FUNCTION_BLOCK MoveMod IMPLEMENTS I_MoveMod
VAR
	mcMoveMod : MC_MoveModulo;
END_VAR
VAR_IN_OUT
	Axis : AXIS_REF;
END_VAR

mcMoveMod(Axis := Axis);

PROPERTY Acceleration : MC_LREAL
GET
Acceleration := mcMoveMod.Acceleration;
END_GET
SET
mcMoveMod.Acceleration := Acceleration;
END_SET
END_PROPERTY

PROPERTY BufferMode : MC_Buffermode
GET
BufferMode := mcMoveMod.BufferMode;
END_GET
SET
mcMoveMod.BufferMode := BufferMode;
END_SET
END_PROPERTY

PROPERTY Busy : BOOL
GET
Busy := mcMoveMod.Busy;
END_GET
END_PROPERTY

PROPERTY Deceleration : MC_LREAL
GET
Deceleration := mcMoveMod.Deceleration;
END_GET
SET
mcMoveMod.Deceleration := Deceleration;
END_SET
END_PROPERTY

PROPERTY Done : BOOL
GET
Done := mcMoveMod.Done;
END_GET
END_PROPERTY

PROPERTY Error : BOOL
GET
Error := mcMoveMod.Error;
END_GET
END_PROPERTY

PROPERTY Execute : BOOL
GET
Execute := mcMoveMod.Execute;
END_GET
SET
mcMoveMod.Execute := Execute;
END_SET
END_PROPERTY

PROPERTY Jerk : MC_LREAL
GET
Jerk := mcMoveMod.Jerk;
END_GET
SET
mcMoveMod.Jerk := Jerk;
END_SET
END_PROPERTY

PROPERTY Position : MC_LREAL
GET
Position := mcMoveMod.Position;
END_GET
SET
mcMoveMod.Position := Position;
END_SET
END_PROPERTY

PROPERTY Velocity : MC_LREAL
GET
Velocity := mcMoveMod.Velocity;
END_GET
SET
mcMoveMod.Velocity := Velocity;
END_SET
END_PROPERTY

END_FUNCTION_BLOCK

(* stored: Version 1.1.0.1
   POU MoveMod: Id {1bfd3278-afcc-4c3c-bae2-f1c6b30d8866}, SpecialFunc None
   Property Acceleration: Id {0d596a7e-59a4-4ff1-b65d-5147cb01f504}
   Get Get: Id {fa6a6f62-d27e-4c07-bef8-33f473fbbcdf}
   Set Set: Id {bec1acfe-50dd-4e03-b13f-0075cdea64fe}
   Property BufferMode: Id {383aa336-aecf-4729-be5a-4928a876364b}
   Get Get: Id {476d401d-a9d7-49ed-8580-9ec8f334d596}
   Set Set: Id {c3669d7b-b91c-4b87-9cbc-09ce1123b73b}
   Property Busy: Id {4f906338-2c35-4182-8130-4b088126df2e}
   Get Get: Id {e2677317-bb42-4496-8737-fc1a199be176}
   Property Deceleration: Id {23702022-baef-491d-8e8a-39565a6c0db1}
   Get Get: Id {41cffb6c-884b-4af2-97ef-8c9ceeb6ee4d}
   Set Set: Id {aeb20737-4404-4eed-9314-f137f39cb149}
   Property Done: Id {9d49c45d-888f-4f5f-abe7-ea7dcff52795}
   Get Get: Id {4d1d556f-75ae-457f-a49c-79d62f4cc6e4}
   Property Error: Id {a092da43-f5c5-4fc3-9ad4-9f21a689b071}
   Get Get: Id {ec2bddf4-5474-4cf0-86db-2bcd939479ee}
   Property Execute: Id {6729b1eb-82a3-4bec-ac1a-aed1fbe49052}
   Get Get: Id {7614de87-20d3-4733-995e-df3b16396c9e}
   Set Set: Id {c7fb56e5-7530-4953-974a-30bb8a162548}
   Property Jerk: Id {1dfb9313-e978-46a2-a93b-14d64bbdd93e}
   Get Get: Id {dd16343b-3036-4d2c-a8eb-64bab3590434}
   Set Set: Id {ee01a914-c076-4eb4-97d0-bce7cca76172}
   Property Position: Id {7c12b022-2f2b-4f2b-b8ee-e4ff0a495548}
   Get Get: Id {39ffb0f6-b656-445c-a80a-557075a93232}
   Set Set: Id {9adab8d2-9008-44dc-9e2c-3d171b4e9df4}
   Property Velocity: Id {121742a5-e664-4c8c-a747-113305b3f1e8}
   Get Get: Id {5fe2da61-9dbb-4408-935d-892fb39e9bcf}
   Set Set: Id {136ff6ca-566c-480a-a4e2-f438a15ee809} *)
